(* PLC project Embox Function Blocks, Embox Embox Function Blocks 1.0 *)
(* stored: creationDateTime 2023-04-26T04:54:00, modificationDateTime 2023-04-26T04:54:00 *)

(* LED_ON *)
FUNCTION_BLOCK LED_ON
  VAR_INPUT
    LED : UINT;  (* LED *)
  END_VAR
  VAR_OUTPUT
    SUCCESS : BOOL;  (* SUCCESS *)
  END_VAR

  SUCCESS := 0;
END_FUNCTION_BLOCK

(* LED_OFF *)
FUNCTION_BLOCK LED_OFF
  VAR_INPUT
    LED : UINT;  (* LED *)
  END_VAR
  VAR_OUTPUT
    SUCCESS : BOOL;  (* SUCCESS *)
  END_VAR

  SUCCESS := 0;
END_FUNCTION_BLOCK
